FUNCTION_BLOCK SyncedSquareWaves EXTENDS CyclicComponent IMPLEMENTS I_Initializable
VAR
	_Initialized  : BOOL;
	PLC_CycleTime : UDINT;
	CycleTime_ms  : LREAL;

	//
	{attribute 'hide'}
	_Wave_500Hz : BOOL;
	{attribute 'hide'}
	_Wave_100Hz : BOOL;
	{attribute 'hide'}
	_Wave_50Hz : BOOL;
	{attribute 'hide'}
	_Wave_5Hz : BOOL;
	{attribute 'hide'}
	_Wave_2Hz : BOOL;
	{attribute 'hide'}
	_Wave_1Hz : BOOL;
	{attribute 'hide'}
	_Wave_0_5Hz : BOOL;
END_VAR

//! @summary This method serves as the entry point for all underlying FB logic
METHOD PUBLIC CyclicLogic
VAR
	Counter		   : LREAL;
	CountsRequired : LREAL;
	CycleCount	   : UDINT;
END_VAR
IF NOT _Initialized THEN
	Initialize();
	RETURN;
END_IF

CycleCount := TwinCAT_SystemInfoVarList._TaskInfo[GETCURTASKINDEXEX()].CycleCount;
IF (CycleTime_ms <= 1) AND (FRAC(1 / CycleTime_ms) = 0) THEN
	CountsRequired := 1 / CycleTime_ms;
	Counter		   := LMOD(CycleCount, CountsRequired);
	IF (Counter + 1) = CountsRequired THEN
		_Wave_500Hz := NOT _Wave_500Hz;
	END_IF
END_IF

IF (CycleTime_ms <= 5) AND (FRAC(5 / CycleTime_ms) = 0) THEN
	CountsRequired := 5 / CycleTime_ms;
	Counter		   := LMOD(CycleCount, CountsRequired);
	IF (Counter + 1) = CountsRequired THEN
		_Wave_100Hz := NOT _Wave_100Hz;
	END_IF
END_IF

IF (CycleTime_ms <= 10) AND (FRAC(10 / CycleTime_ms) = 0) THEN
	CountsRequired := 10 / CycleTime_ms;
	Counter		   := LMOD(CycleCount, CountsRequired);
	IF (Counter + 1) = CountsRequired THEN
		_Wave_50Hz := NOT _Wave_50Hz;
	END_IF
END_IF

IF (CycleTime_ms <= 100) AND (FRAC(100 / CycleTime_ms) = 0) THEN
	CountsRequired := 100 / CycleTime_ms;
	Counter		   := LMOD(CycleCount, CountsRequired);
	IF (Counter + 1) = CountsRequired THEN
		_Wave_5Hz := NOT _Wave_5Hz;
	END_IF
END_IF

IF (CycleTime_ms <= 250) AND (FRAC(250 / CycleTime_ms) = 0) THEN
	CountsRequired := 250 / CycleTime_ms;
	Counter		   := LMOD(CycleCount, CountsRequired);
	IF (Counter + 1) = CountsRequired THEN
		_Wave_2Hz := NOT _Wave_2Hz;
	END_IF
END_IF

IF (CycleTime_ms <= 500) AND (FRAC(500 / CycleTime_ms) = 0) THEN
	CountsRequired := 500 / CycleTime_ms;
	Counter		   := LMOD(CycleCount, CountsRequired);
	IF (Counter + 1) = CountsRequired THEN
		_Wave_1Hz := NOT _Wave_1Hz;
	END_IF
END_IF

IF (CycleTime_ms <= 1000) AND (FRAC(1000 / CycleTime_ms) = 0) THEN
	CountsRequired := 1000 / CycleTime_ms;
	Counter		   := LMOD(CycleCount, CountsRequired);
	IF (Counter + 1) = CountsRequired THEN
		_Wave_0_5Hz := NOT _Wave_0_5Hz;
	END_IF
END_IF
END_METHOD

METHOD Initialize
//PLC Scan Info
PLC_CycleTime := TwinCAT_SystemInfoVarList._TaskInfo[GETCURTASKINDEXEX()].CycleTime;
CycleTime_ms  := TO_LREAL(PLC_CycleTime) / 10000.0;

//
_Wave_500Hz	 := TRUE;
_Wave_100Hz	 := TRUE;
_Wave_50Hz	 := TRUE;
_Wave_5Hz	 := TRUE;
_Wave_2Hz	 := TRUE;
_Wave_1Hz	 := TRUE;
_Wave_0_5Hz	 := TRUE;
_Initialized := TRUE;
END_METHOD

{attribute 'monitoring' := 'call'}
PROPERTY Initialized : BOOL
GET
Initialized := _Initialized;
END_GET
SET
_Initialized := Initialized;
END_SET
END_PROPERTY

{attribute 'monitoring' := 'call'}
PROPERTY Wave_0_5Hz : BOOL
GET
Wave_0_5Hz := _Wave_0_5Hz;
END_GET
END_PROPERTY

{attribute 'monitoring' := 'call'}
PROPERTY Wave_100Hz : BOOL
GET
Wave_100Hz := _Wave_100Hz;
END_GET
END_PROPERTY

{attribute 'monitoring' := 'call'}
PROPERTY Wave_1Hz : BOOL
GET
Wave_1Hz := _Wave_1Hz;
END_GET
END_PROPERTY

{attribute 'monitoring' := 'call'}
PROPERTY Wave_2Hz : BOOL
GET
Wave_2Hz := _Wave_2Hz;
END_GET
END_PROPERTY

{attribute 'monitoring' := 'call'}
PROPERTY Wave_500Hz : BOOL
GET
Wave_500Hz := _Wave_500Hz;
END_GET
END_PROPERTY

{attribute 'monitoring' := 'call'}
PROPERTY Wave_50Hz : BOOL
GET
Wave_50Hz := _Wave_50Hz;
END_GET
END_PROPERTY

{attribute 'monitoring' := 'call'}
PROPERTY Wave_5Hz : BOOL
GET
Wave_5Hz := _Wave_5Hz;
END_GET
END_PROPERTY

END_FUNCTION_BLOCK

(* stored: Version 1.1.0.1, ProductVersion 3.1.4026.18
   POU SyncedSquareWaves: Id {35f66174-c5b3-49ca-9765-0f46a12be9be}, SpecialFunc None
   Folder Initializable: Id {d2affa53-c5ae-459e-a173-712d2ffbc097}
   Method CyclicLogic: Id {5e3838da-f4d8-4716-ac0d-b7b9f9f0dadb}
   Method Initialize: Id {b0d4565e-7f87-4a88-8840-de4c795a7bf2}
   Property Initialized: Id {7d30abb5-9e0b-4781-ba98-53b2bfac6182}
   Get Get: Id {d08c54b2-51c3-4edc-ad2d-83328c965cc3}
   Set Set: Id {9f368cae-4e7a-47a7-820f-08d192fff5b3}
   Property Wave_0_5Hz: Id {fd3d835b-3d2a-4fc5-8158-9a11dac255e3}
   Get Get: Id {c1d46175-9e18-4011-a083-dbff3549dd73}
   Property Wave_100Hz: Id {b64fcb53-b055-452e-9663-c4625a169b20}
   Get Get: Id {9fc00187-6221-4d6d-a1d4-a510f39f14fe}
   Property Wave_1Hz: Id {01d8919c-b328-49b5-a235-50ecde21edf8}
   Get Get: Id {78e216e5-2c86-447d-bdba-220b6e0ae890}
   Property Wave_2Hz: Id {8d052cca-5f43-4ed2-a3df-764c43e95820}
   Get Get: Id {31e3ad99-a798-4f3c-8553-59c87de98b80}
   Property Wave_500Hz: Id {ee378a0f-1e3a-4791-99da-444ed1ab3b8f}
   Get Get: Id {2bad6ca2-5441-4f2e-979c-97f31de408cc}
   Property Wave_50Hz: Id {3d42c34c-0bd9-4b99-8a94-4b7443d1ba08}
   Get Get: Id {e74ab5f7-0350-4d60-94cf-e6771e185218}
   Property Wave_5Hz: Id {7ac74df0-a221-4a97-8491-dfa3c586e258}
   Get Get: Id {5232fbab-6bcc-418f-abfa-2ccb6cb1a396} *)
